FUNCTION_BLOCK TimeOutMovement (* Basic FB with empty ECC *)
  (* Standard: 61499-2 *)
  (* Version 1.0, 2023-03-16, AK125171 *)
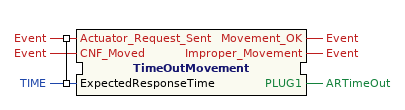
  EVENT_INPUT
    Actuator_Request_Sent WITH ExpectedResponseTime;
    CNF_Moved;
  END_EVENT
  EVENT_OUTPUT
    Movement_OK;
    Improper_Movement;
  END_EVENT
  VAR_INPUT
    ExpectedResponseTime : TIME;
  END_VAR
  PLUGS
    PLUG1 : ARTimeOut;
  END_PLUGS
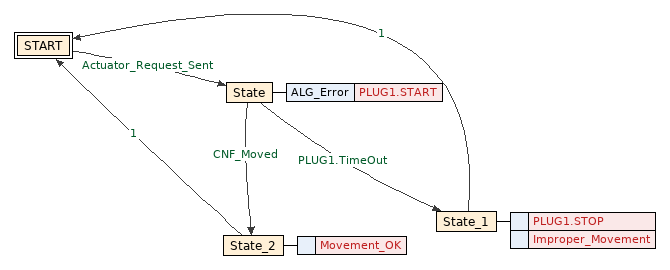
  EC_STATES
    START; (* Initial State *)
    State : ALG_Error -> PLUG1.START;
    State_1 : -> PLUG1.STOP, -> Improper_Movement;
    State_2 : -> Movement_OK;
  END_STATES
  EC_TRANSITIONS
    START TO State := Actuator_Request_Sent;
    State TO State_1 := PLUG1.TimeOut;
    State_1 TO START := 1;
    State TO State_2 := CNF_Moved;
    State_2 TO START := 1;
  END_TRANSITIONS
  ALGORITHM ALG_Error IN ST:
Plug1.DT:=ExpectedResponseTime;
  END_ALGORITHM
END_FUNCTION_BLOCK
